Fanuc KAREL source: kb00070.KL

-- PROVISIONAL review KL for V1013-1; original PC SHA256 7c443d78c82385fd1e734d6fcf15355169f0995435031029170dfa8cac776ba9
-- Incomplete behavior may be omitted. Consult companion uncertainty JSON. Do not deploy.
PROGRAM KB00070
%NOLOCKGROUP
BEGIN
  -- UNRESOLVED_PC offsets 5-12; opcodes 9D,23
  -- UNRESOLVED_PC offsets 17-24; opcodes 9D,23
  -- UNRESOLVED_PC offsets 29-38; opcodes 3F,75
  -- UNRESOLVED_PC offsets 43-50; opcodes 9D,23
  -- UNRESOLVED_PC offsets 55-64; opcodes 3F,75
  -- UNRESOLVED_PC offsets 69-76; opcodes 9D,23
  -- UNRESOLVED_PC offsets 81-88; opcodes 9D,23
  -- UNRESOLVED_PC offsets 93-102; opcodes 3F,75
  -- UNRESOLVED_PC offsets 107-165; opcodes 27,22,22,22,2A,22,22,2A,22,22,22,2A,31
  -- UNRESOLVED_PC offsets 170-174; opcodes 7F
END KB00070
